// TIA Portal V16 export
// export: Created 2022-02-04T14:40:20.6333267Z, ExportSetting WithDefaults, DisplayName Totally Integrated Automation Portal, DisplayVersion V16 Update 1, DisplayName TIA Portal Version Control Interface, DisplayVersion V16, DisplayName TIA Portal Openness, DisplayVersion V16, DisplayName SINAMICS Startdrive Advanced, DisplayVersion V16 Update 5, DisplayName SINAMICS Startdrive G130, G150, S120, S150, SINAMICS MV, S210, DisplayVersion V16 Update 5, DisplayName SINAMICS Startdrive G110M, G120, G120C, G120D, G120P, G115D, DisplayVersion V16 Update 5, DisplayName STEP 7 Professional, DisplayVersion V16, DisplayName STEP 7 Safety, DisplayVersion V16, DisplayName WinCC Advanced, DisplayVersion V16, DisplayName SIMATIC Visualization Architect, DisplayVersion V16
DATA_BLOCK "QueueController_DB"   // DB11
AUTHOR : Aspir
VERSION : 0.1
// stored: AutoNumber true, InstanceOfName QueueController, InstanceOfType FB
"QueueController"
   // VAR_INPUT
   //    Reset : Bool;
   //    ResetSxema : Bool;
   //    NoChessLayout : Bool;
   //    CheckPlankL : Bool;
   //    ChainInd : Bool;
   //    Hole : Bool;
   //    Done : Bool;
   //    Length : Int;
   //    CheckL : Int;
   //    PT : Int;
   //    plankW : Int;
   //    plankT : Int;
   //    OffsetBB : Int;
   // END_VAR
   // VAR_OUTPUT
   //    CommonSxemaAlarm : Bool;
   //    AlarmNotAwaitableBoard : Bool;
   //    AlarmNotValidHole : Bool;
   //    AlarmCount : Bool;
   //    AlarmWrongLength : Bool;
   //    Hint_1 : Bool;
   //    Hint_2 : Bool;
   //    Hint_3 : Bool;
   //    CorrectingCounters : Bool;
   //    CorrectCounters : Bool;
   //    CorrectWheel : Bool;
   //    GettingLastLay : Bool;
   //    CurrentLayCounter : Int;
   // END_VAR
   // VAR_IN_OUT
   //    BoardsInLay_counter : Int;
   //    Layer_Volume { ExternalAccessible := 'False'; ExternalVisible := 'False'; ExternalWritable := 'False'} : DInt;
   // END_VAR
   // VAR RETAIN
   //    Calibrated : Bool;
   //    AwaitedChain : Bool;
   //    AwaitEmptySpace : Bool;
   //    ProcessedError : Bool;
   //    CanPutBoardHoleBefore : Bool;
   //    LugCounter : Int;
   //    Data : Array[0..15] of "PlankOnChain";
   // END_VAR
BEGIN
END_DATA_BLOCK
